(* CoDeSys 2.3 export: Rtu11word7SJ6xm0.EXP *)

(* POU SGL_Sismored/Sismored 4.0/Imported/Rtu11word7SJ6xm0, FAI *)
FUNCTION_BLOCK Rtu11word7SJ6xm0
VAR_INPUT
    xFirstCycle : BOOL;
    iSequenceOrder: INT;
    sProtocol: STRING;
    eState: eStates;
    eAction: eActions;
    wInput1, wInput2, wInput3, wInput4, wInput5, wInput6, wInput7, wInput8, wInput9, wInput10, wInput11: WORD;
                                                                                           (*input signals*)
    xSave1, xSave2, xSave3, xSave4, xSave5, xSave6, xSave7, xSave8, xSave9, xSave10, xSave11 : BOOL;                                                                             (*save signals*)
    sName1, sName2, sName3, sName4, sName5, sName6, sName7, sName8, sName9, sName10, sName11 : STRING;                                                                         (*name signals*)
                                                                                               (*status com*)
END_VAR
VAR_OUTPUT
                                                                                               (*output signals*)
    wOutput1, wOutput2, wOutput3, wOutput4, wOutput5, wOutput6, wOutput7, wOutput8, wOutput9, wOutput10, wOutput11: WORD;
                                                                                           (*select*)
                                                                                               (*execute*)
END_VAR
VAR
                                                                                          (*instances*)
    sTime: STRING;
    aSignals : ARRAY[1..inst0Map11word7SJ6xm0 : Map11word7SJ6xm0;
inst0Pack11word7SJ6xm0 : Pack11word7SJ6xm0;
inst0Pack11bool7SJ6xm0 : Pack11bool7SJ6xm0;
inst0Pack11string7SJ6xm0 : Pack11string7SJ6xm0;
inst0Check11word7SJ6xm0 : Check11word7SJ6xm0;
] OF 11;                                      (*number of signals | data type*)
    aMaskChanges : ARRAY[1..WORD] OF BOOL;                  (*number of signals*)
    aNames : ARRAY[1..11] OF STRING;                           (*number of signals*)
    aSaves : ARRAY[1..11] OF BOOL;                                 (*number of signals*)
    11                                                                                      (*sbo internal variables*)
END_VAR
(* body not read: x-want_COMMENT *)
END_FUNCTION_BLOCK
